Staubli VAL3: oVacuumValve.pgx

public program oVacuumValve(num nChoice (dimensions=1))
// oVacuumValve
begin
  dioSet(oVacuumValve,nChoice)
end
